{attribute 'GeneratedUsingTerminal: EL2202-0000-0016'}
{attribute addProperty BoxType "EL2202-0000-0016"}
{attribute addProperty Id "EtcSlaveTerminalBaseChannel_1AT %Q*Channel_54BE63B32Channel_2AT %Q*Channel_54BE63B32WcStateAT %I*WcState_0B2B16F91InfoDataAT %I*InfoData_6F19DB2B2"}
{attribute addProperty CRC "1985922692"}
{attribute addProperty Size "7"}
TYPE EL2202_765EC684 EXTENDS EtcSlaveTerminalBase :
STRUCT
	{attribute addProperty Name "Channel_1"}
	Channel_1 : Channel_54BE63B3;
	{attribute addProperty Name "Channel_2"}
	Channel_2 : Channel_54BE63B3;
	{attribute addProperty Name "WcState"}
	WcState : WcState_0B2B16F9;
	{attribute addProperty Name "InfoData"}
	InfoData : InfoData_6F19DB2B;
END_STRUCT
END_TYPE

(* stored: Version 1.2.0.0, ProductVersion 3.1.4024.9
   DUT EL2202_765EC684: Id {20762b9b-234a-4bc6-98d2-d4a874c1736e} *)
